LIN {X 0,Y 92.018,Z 344.154,A -85,B 0,C 180,E1 -28315.718,E2 -28315.718} C_VEL
LIN {X 0,Y 86.368,Z 354.698,A -85,B 0,C 180,E1 -28320.776,E2 -28320.776} C_VEL
LIN {X 0,Y 80.821,Z 363.839,A -85,B 0,C 180,E1 -28326.964,E2 -28326.964} C_VEL
LIN {X 0,Y 76.179,Z 371.216,A -85,B 0,C 180,E1 -28333.933,E2 -28333.933} C_VEL
LIN {X 0,Y 72.82,Z 377.117,A -85,B 0,C 180,E1 -28341.676,E2 -28341.676} C_VEL
LIN {X 0,Y 70.618,Z 381.782,A -85,B 0,C 180,E1 -28350,E2 -28350} C_VEL
LIN {X 0,Y 70.293,Z 382.581,A -85,B 0,C 180,E1 -28351.768,E2 -28351.768} C_VEL
LIN {X 0,Y 68.904,Z 384.476,A -85,B 0,C 180,E1 -28356.25,E2 -28356.25} C_VEL
LIN {X 0,Y 65.683,Z 386.983,A -85,B 0,C 180,E1 -28363.945,E2 -28363.945} C_VEL
LIN {X 0,Y 63.762,Z 388.494,A -85,B 0,C 180,E1 -28370.668,E2 -28370.668} C_VEL
LIN {X 0,Y 63.611,Z 389.367,A -85,B 0,C 180,E1 -28375.957,E2 -28375.957} C_VEL
LIN {X 0,Y 63.921,Z 389.596,A -85,B 0,C 180,E1 -28377.701,E2 -28377.701} C_VEL
LIN {X 0,Y 67.759,Z 390.402,A -85,B 0,C 180,E1 -28388.485,E2 -28388.485} C_VEL
LIN {X 0,Y 73.771,Z 389.834,A -85,B 0,C 180,E1 -28398.183,E2 -28398.183} C_VEL
LIN {X 0,Y 78.574,Z 388.718,A -85,B 0,C 180,E1 -28403.608,E2 -28403.608} C_VEL
LIN {X 0,Y 83.148,Z 387.318,A -85,B 0,C 180,E1 -28407.695,E2 -28407.695} C_VEL
LIN {X 0,Y 90.439,Z 384.448,A -85,B 0,C 180,E1 -28412.842,E2 -28412.842} C_VEL
LIN {X 0,Y 98.878,Z 380.236,A -85,B 0,C 180,E1 -28417.515,E2 -28417.515} C_VEL
LIN {X 0,Y 107.812,Z 374.74,A -85,B 0,C 180,E1 -28421.393,E2 -28421.393} C_VEL
LIN {X 0,Y 108.744,Z 373.558,A -85,B 0,C 180,E1 -28423.099,E2 -28423.099} C_VEL
LIN {X 0,Y 109.834,Z 371.724,A -85,B 0,C 180,E1 -28426.233,E2 -28426.233} C_VEL
LIN {X 0,Y 110.579,Z 370.301,A -85,B 0,C 180,E1 -28429.013,E2 -28429.013} C_VEL
LIN {X 0,Y 111.224,Z 368.711,A -85,B 0,C 180,E1 -28432.744,E2 -28432.744} C_VEL
LIN {X 0,Y 111.839,Z 367.436,A -85,B 0,C 180,E1 -28436.401,E2 -28436.401} C_VEL
LIN {X 0,Y 112.278,Z 366.529,A -85,B 0,C 180,E1 -28440.004,E2 -28440.004} C_VEL
LIN {X 0,Y 112.294,Z 366.253,A -85,B 0,C 180,E1 -28443.593,E2 -28443.593} C_VEL
LIN {X 0,Y 111.927,Z 366.629,A -85,B 0,C 180,E1 -28447.219,E2 -28447.219} C_VEL
LIN {X 0,Y 111.564,Z 367.372,A -85,B 0,C 180,E1 -28450.898,E2 -28450.898} C_VEL
LIN {X 0,Y 111.237,Z 368.424,A -85,B 0,C 180,E1 -28454.643,E2 -28454.643} C_VEL
LIN {X 0,Y 110.286,Z 370.941,A -85,B 0,C 180,E1 -28460.522,E2 -28460.522} C_VEL
LIN {X 0,Y 108.905,Z 373.784,A -85,B 0,C 180,E1 -28465.386,E2 -28465.386} C_VEL
LIN {X 0,Y 107.482,Z 376.257,A -85,B 0,C 180,E1 -28469.068,E2 -28469.068} C_VEL
LIN {X 0,Y 106.076,Z 377.68,A -85,B 0,C 180,E1 -28470.539,E2 -28470.539} C_VEL
LIN {X 0,Y 100.57,Z 381.248,A -85,B 0,C 180,E1 -28473.012,E2 -28473.012} C_VEL
LIN {X 0,Y 92.528,Z 385.67,A -85,B 0,C 180,E1 -28477.107,E2 -28477.107} C_VEL
LIN {X 0,Y 85.091,Z 389.05,A -85,B 0,C 180,E1 -28481.984,E2 -28481.984} C_VEL
LIN {X 0,Y 76.184,Z 392.05,A -85,B 0,C 180,E1 -28489.78,E2 -28489.78} C_VEL
LIN {X 0,Y 69.088,Z 393.493,A -85,B 0,C 180,E1 -28499.429,E2 -28499.429} C_VEL
LIN {X 0,Y 64.576,Z 393.358,A -85,B 0,C 180,E1 -28510.944,E2 -28510.944} C_VEL
LIN {X 0,Y 62.726,Z 391.712,A -85,B 0,C 180,E1 -28523.567,E2 -28523.567} C_VEL
LIN {X 0,Y 62.679,Z 390.242,A -85,B 0,C 180,E1 -28530,E2 -28530} C_VEL
LIN {X 0,Y 62.887,Z 387.196,A -85,B 0,C 180,E1 -28539.65,E2 -28539.65} C_VEL
LIN {X 0,Y 64.422,Z 383.057,A -85,B 0,C 180,E1 -28549.104,E2 -28549.104} C_VEL
LIN {X 0,Y 68.042,Z 376.693,A -85,B 0,C 180,E1 -28559.381,E2 -28559.381} C_VEL
LIN {X 0,Y 72.677,Z 369.751,A -85,B 0,C 180,E1 -28567.184,E2 -28567.184} C_VEL
LIN {X 0,Y 77.715,Z 361.895,A -85,B 0,C 180,E1 -28573.522,E2 -28573.522} C_VEL
LIN {X 0,Y 81.578,Z 355.857,A -85,B 0,C 180,E1 -28577.077,E2 -28577.077} C_VEL
LIN {X 0,Y 85.122,Z 346.402,A -85,B 0,C 180,E1 -28582.623,E2 -28582.623} C_VEL
LIN {X 0,Y 87.485,Z 337.692,A -85,B 0,C 180,E1 -28587.157,E2 -28587.157} C_VEL
LIN {X 0,Y 87.648,Z 335.398,A -85,B 0,C 180,E1 -28588.581,E2 -28588.581} C_VEL
LIN {X 0,Y 87.041,Z 330.108,A -85,B 0,C 180,E1 -28592.643,E2 -28592.643} C_VEL
LIN {X 0,Y 86.061,Z 326.798,A -85,B 0,C 180,E1 -28595.895,E2 -28595.895} C_VEL
LIN {X 0,Y 85.319,Z 324.626,A -85,B 0,C 180,E1 -28598.237,E2 -28598.237} C_VEL
LIN {X 0,Y 83.779,Z 321.175,A -85,B 0,C 180,E1 -28602.92,E2 -28602.92} C_VEL
LIN {X 0,Y 81.877,Z 316.988,A -85,B 0,C 180,E1 -28610.109,E2 -28610.109} C_VEL
LIN {X 0,Y 80.619,Z 314.216,A -85,B 0,C 180,E1 -28617.496,E2 -28617.496} C_VEL
LIN {X 0,Y 80.581,Z 313.017,A -85,B 0,C 180,E1 -28619.994,E2 -28619.994} C_VEL
LIN {X 0,Y 80.065,Z 312.777,A -85,B 0,C 180,E1 -28626.992,E2 -28626.992} C_VEL
LIN {X 0,Y 80.116,Z 312.914,A -85,B 0,C 180,E1 -28630.098,E2 -28630.098} C_VEL
LIN {X 0,Y 80.243,Z 314.44,A -85,B 0,C 180,E1 -28635.55,E2 -28635.55} C_VEL
LIN {X 0,Y 81.919,Z 317.887,A -85,B 0,C 180,E1 -28645.395,E2 -28645.395} C_VEL
LIN {X 0,Y 83.202,Z 320.714,A -85,B 0,C 180,E1 -28650.445,E2 -28650.445} C_VEL
LIN {X 0,Y 85.06,Z 325.54,A -85,B 0,C 180,E1 -28656.884,E2 -28656.884} C_VEL
LIN {X 0,Y 86.237,Z 328.978,A -85,B 0,C 180,E1 -28660.682,E2 -28660.682} C_VEL
LIN {X 0,Y 87.697,Z 334.701,A -85,B 0,C 180,E1 -28666.15,E2 -28666.15} C_VEL
LIN {X 0,Y 88.081,Z 336.72,A -85,B 0,C 180,E1 -28667.886,E2 -28667.886} C_VEL
LIN {X 0,Y 87.681,Z 340.216,A -85,B 0,C 180,E1 -28670.117,E2 -28670.117} C_VEL
LIN {X 0,Y 86.704,Z 344.364,A -85,B 0,C 180,E1 -28672.561,E2 -28672.561} C_VEL
LIN {X 0,Y 81.324,Z 353.994,A -85,B 0,C 180,E1 -28677.308,E2 -28677.308} C_VEL
LIN {X 0,Y 76.185,Z 361.944,A -85,B 0,C 180,E1 -28682.533,E2 -28682.533} C_VEL
LIN {X 0,Y 70.878,Z 369.719,A -85,B 0,C 180,E1 -28689.694,E2 -28689.694} C_VEL
LIN {X 0,Y 66.874,Z 375.937,A -85,B 0,C 180,E1 -28697.867,E2 -28697.867} C_VEL
LIN {X 0,Y 64.091,Z 380.892,A -85,B 0,C 180,E1 -28706.857,E2 -28706.857} C_VEL
LIN {X 0,Y 62.438,Z 384.742,A -85,B 0,C 180,E1 -28716.462,E2 -28716.462} C_VEL
LIN {X 0,Y 62.098,Z 386.739,A -85,B 0,C 180,E1 -28723.082,E2 -28723.082} C_VEL
LIN {X 0,Y 62.492,Z 388.303,A -85,B 0,C 180,E1 -28729.717,E2 -28729.717} C_VEL
LIN {X 0,Y 63.921,Z 389.596,A -85,B 0,C 180,E1 -28737.701,E2 -28737.701} C_VEL
LIN {X 0,Y 64.741,Z 390.181,A -85,B 0,C 180,E1 -28742.889,E2 -28742.889} C_VEL
LIN {X 0,Y 65.462,Z 390.63,A -85,B 0,C 180,E1 -28751.598,E2 -28751.598} C_VEL
LIN {X 0,Y 66.926,Z 390.437,A -85,B 0,C 180,E1 -28758.374,E2 -28758.374} C_VEL
LIN {X 0,Y 69.282,Z 389.92,A -85,B 0,C 180,E1 -28762.928,E2 -28762.928} C_VEL
LIN {X 0,Y 70.378,Z 389.67,A -85,B 0,C 180,E1 -28764.26,E2 -28764.26} C_VEL
LIN {X 0,Y 74.417,Z 388.783,A -85,B 0,C 180,E1 -28768.205,E2 -28768.205} C_VEL
LIN {X 0,Y 84.112,Z 385.635,A -85,B 0,C 180,E1 -28775.312,E2 -28775.312} C_VEL
LIN {X 0,Y 93.339,Z 381.565,A -85,B 0,C 180,E1 -28780.248,E2 -28780.248} C_VEL
LIN {X 0,Y 102.448,Z 376.503,A -85,B 0,C 180,E1 -28784.079,E2 -28784.079} C_VEL
LIN {X 0,Y 103.419,Z 375.35,A -85,B 0,C 180,E1 -28786.245,E2 -28786.245} C_VEL
LIN {X 0,Y 104.064,Z 374.379,A -85,B 0,C 180,E1 -28788.316,E2 -28788.316} C_VEL
LIN {X 0,Y 105.039,Z 372.811,A -85,B 0,C 180,E1 -28792.315,E2 -28792.315} C_VEL
LIN {X 0,Y 105.802,Z 371.552,A -85,B 0,C 180,E1 -28796.196,E2 -28796.196} C_VEL
LIN {X 0,Y 106.434,Z 370.677,A -85,B 0,C 180,E1 -28800.005,E2 -28800.005} C_VEL
LIN {X 0,Y 106.488,Z 370.442,A -85,B 0,C 180,E1 -28803.789,E2 -28803.789} C_VEL
LIN {X 0,Y 106.069,Z 370.864,A -85,B 0,C 180,E1 -28807.62,E2 -28807.62} C_VEL
LIN {X 0,Y 105.594,Z 371.64,A -85,B 0,C 180,E1 -28811.522,E2 -28811.522} C_VEL
LIN {X 0,Y 105.046,Z 372.775,A -85,B 0,C 180,E1 -28815.527,E2 -28815.527} C_VEL
LIN {X 0,Y 104.295,Z 374.396,A -85,B 0,C 180,E1 -28819.695,E2 -28819.695} C_VEL
LIN {X 0,Y 102.829,Z 376.705,A -85,B 0,C 180,E1 -28824.215,E2 -28824.215} C_VEL
LIN {X 0,Y 101.948,Z 377.966,A -85,B 0,C 180,E1 -28826.342,E2 -28826.342} C_VEL
LIN {X 0,Y 99.787,Z 379.719,A -85,B 0,C 180,E1 -28828.315,E2 -28828.315} C_VEL
LIN {X 0,Y 91.18,Z 384.423,A -85,B 0,C 180,E1 -28832.023,E2 -28832.023} C_VEL
LIN {X 0,Y 84.735,Z 387.375,A -85,B 0,C 180,E1 -28835.499,E2 -28835.499} C_VEL
LIN {X 0,Y 75.513,Z 390.701,A -85,B 0,C 180,E1 -28841.881,E2 -28841.881} C_VEL
LIN {X 0,Y 66.722,Z 392.85,A -85,B 0,C 180,E1 -28850.804,E2 -28850.804} C_VEL
LIN {X 0,Y 63.056,Z 393.309,A -85,B 0,C 180,E1 -28856.133,E2 -28856.133} C_VEL
LIN {X 0,Y 57.893,Z 393.106,A -85,B 0,C 180,E1 -28868.643,E2 -28868.643} C_VEL
LIN {X 0,Y 56.396,Z 392.443,A -85,B 0,C 180,E1 -28875.568,E2 -28875.568} C_VEL
LIN {X 0,Y 55.663,Z 391.363,A -85,B 0,C 180,E1 -28882.747,E2 -28882.747} C_VEL
LIN {X 0,Y 55.589,Z 389.853,A -85,B 0,C 180,E1 -28890,E2 -28890} C_VEL
LIN {X 0,Y 55.885,Z 386.73,A -85,B 0,C 180,E1 -28900.873,E2 -28900.873} C_VEL
LIN {X 0,Y 57.705,Z 382.508,A -85,B 0,C 180,E1 -28911.43,E2 -28911.43} C_VEL
LIN {X 0,Y 61.928,Z 376.062,A -85,B 0,C 180,E1 -28922.619,E2 -28922.619} C_VEL
LIN {X 0,Y 67.111,Z 369.001,A -85,B 0,C 180,E1 -28930.882,E2 -28930.882} C_VEL
LIN {X 0,Y 72.955,Z 360.676,A -85,B 0,C 180,E1 -28937.589,E2 -28937.589} C_VEL
LIN {X 0,Y 75.706,Z 356.698,A -85,B 0,C 180,E1 -28939.983,E2 -28939.983} C_VEL
LIN {X 0,Y 79.215,Z 348.739,A -85,B 0,C 180,E1 -28945.013,E2 -28945.013} C_VEL
LIN {X 0,Y 82.21,Z 339.886,A -85,B 0,C 180,E1 -28950.006,E2 -28950.006} C_VEL
LIN {X 0,Y 82.184,Z 335.431,A -85,B 0,C 180,E1 -28953.632,E2 -28953.632} C_VEL
LIN {X 0,Y 81.547,Z 331.959,A -85,B 0,C 180,E1 -28957.175,E2 -28957.175} C_VEL
LIN {X 0,Y 80.973,Z 329.88,A -85,B 0,C 180,E1 -28959.679,E2 -28959.679} C_VEL
LIN {X 0,Y 79.736,Z 326.561,A -85,B 0,C 180,E1 -28964.661,E2 -28964.661} C_VEL
LIN {X 0,Y 78.714,Z 323.787,A -85,B 0,C 180,E1 -28969.707,E2 -28969.707} C_VEL
LIN {X 0,Y 77.638,Z 319.844,A -85,B 0,C 180,E1 -28979.994,E2 -28979.994} C_VEL
LIN {X 0,Y 77.36,Z 319.227,A -85,B 0,C 180,E1 -28985.206,E2 -28985.206} C_VEL
LIN {X 0,Y 77.248,Z 319.631,A -85,B 0,C 180,E1 -28990.477,E2 -28990.477} C_VEL
LIN {X 0,Y 78.273,Z 323.727,A -85,B 0,C 180,E1 -29003.824,E2 -29003.824} C_VEL
LIN {X 0,Y 79.211,Z 326.244,A -85,B 0,C 180,E1 -29008.91,E2 -29008.91} C_VEL
LIN {X 0,Y 80.712,Z 331.117,A -85,B 0,C 180,E1 -29016.07,E2 -29016.07} C_VEL
LIN {X 0,Y 81.599,Z 334.606,A -85,B 0,C 180,E1 -29020.226,E2 -29020.226} C_VEL
LIN {X 0,Y 82.422,Z 339.119,A -85,B 0,C 180,E1 -29024.919,E2 -29024.919} C_VEL
LIN {X 0,Y 82.541,Z 340.301,A -85,B 0,C 180,E1 -29026.043,E2 -29026.043} C_VEL
LIN {X 0,Y 81.813,Z 343.621,A -85,B 0,C 180,E1 -29028.261,E2 -29028.261} C_VEL
LIN {X 0,Y 81.23,Z 345.605,A -85,B 0,C 180,E1 -29029.542,E2 -29029.542} C_VEL
LIN {X 0,Y 75.424,Z 355.068,A -85,B 0,C 180,E1 -29034.383,E2 -29034.383} C_VEL
LIN {X 0,Y 68.937,Z 364.216,A -85,B 0,C 180,E1 -29041.037,E2 -29041.037} C_VEL
LIN {X 0,Y 63.399,Z 371.597,A -85,B 0,C 180,E1 -29048.883,E2 -29048.883} C_VEL
LIN {X 0,Y 59.904,Z 376.587,A -85,B 0,C 180,E1 -29056.429,E2 -29056.429} C_VEL
LIN {X 0,Y 56.932,Z 381.448,A -85,B 0,C 180,E1 -29066.461,E2 -29066.461} C_VEL
LIN {X 0,Y 55.244,Z 385.213,A -85,B 0,C 180,E1 -29077.308,E2 -29077.308} C_VEL
LIN {X 0,Y 55.029,Z 387.169,A -85,B 0,C 180,E1 -29084.798,E2 -29084.798} C_VEL
LIN {X 0,Y 55.663,Z 388.654,A -85,B 0,C 180,E1 -29092.257,E2 -29092.257} C_VEL
LIN {X 0,Y 57.536,Z 389.922,A -85,B 0,C 180,E1 -29101.252,E2 -29101.252} C_VEL
LIN {X 0,Y 62.136,Z 390.62,A -85,B 0,C 180,E1 -29112.736,E2 -29112.736} C_VEL
LIN {X 0,Y 68.298,Z 390.08,A -85,B 0,C 180,E1 -29121.882,E2 -29121.882} C_VEL
LIN {X 0,Y 70.378,Z 389.67,A -85,B 0,C 180,E1 -29124.26,E2 -29124.26} C_VEL
LIN {X 0,Y 73.522,Z 388.919,A -85,B 0,C 180,E1 -29128.189,E2 -29128.189} C_VEL
LIN {X 0,Y 77.999,Z 387.228,A -85,B 0,C 180,E1 -29134.767,E2 -29134.767} C_VEL
LIN {X 0,Y 82.072,Z 385.454,A -85,B 0,C 180,E1 -29139.487,E2 -29139.487} C_VEL
LIN {X 0,Y 85.943,Z 383.765,A -85,B 0,C 180,E1 -29142.315,E2 -29142.315} C_VEL
LIN {X 0,Y 87.431,Z 383.121,A -85,B 0,C 180,E1 -29143.063,E2 -29143.063} C_VEL
LIN {X 0,Y 94.223,Z 379.862,A -85,B 0,C 180,E1 -29145.843,E2 -29145.843} C_VEL
LIN {X 0,Y 97.267,Z 378.117,A -85,B 0,C 180,E1 -29147.486,E2 -29147.486} C_VEL
LIN {X 0,Y 99.009,Z 376.01,A -85,B 0,C 180,E1 -29153.588,E2 -29153.588} C_VEL
LIN {X 0,Y 99.528,Z 375.344,A -85,B 0,C 180,E1 -29155.956,E2 -29155.956} C_VEL
LIN {X 0,Y 100.325,Z 374.473,A -85,B 0,C 180,E1 -29160.005,E2 -29160.005} C_VEL
LIN {X 0,Y 100.449,Z 374.273,A -85,B 0,C 180,E1 -29164.017,E2 -29164.017} C_VEL
LIN {X 0,Y 99.723,Z 374.978,A -85,B 0,C 180,E1 -29169.38,E2 -29169.38} C_VEL
LIN {X 0,Y 99.306,Z 375.582,A -85,B 0,C 180,E1 -29172.263,E2 -29172.263} C_VEL
LIN {X 0,Y 98.538,Z 376.825,A -85,B 0,C 180,E1 -29176.581,E2 -29176.581} C_VEL
LIN {X 0,Y 97.285,Z 378.592,A -85,B 0,C 180,E1 -29181.179,E2 -29181.179} C_VEL
LIN {X 0,Y 96.033,Z 380.11,A -85,B 0,C 180,E1 -29184.302,E2 -29184.302} C_VEL
LIN {X 0,Y 93.588,Z 381.569,A -85,B 0,C 180,E1 -29185.694,E2 -29185.694} C_VEL
LIN {X 0,Y 84.714,Z 385.821,A -85,B 0,C 180,E1 -29189.416,E2 -29189.416} C_VEL
LIN {X 0,Y 76.289,Z 389.043,A -85,B 0,C 180,E1 -29193.995,E2 -29193.995} C_VEL
LIN {X 0,Y 65.944,Z 391.894,A -85,B 0,C 180,E1 -29201.754,E2 -29201.754} C_VEL
LIN {X 0,Y 57.281,Z 393.126,A -85,B 0,C 180,E1 -29212.161,E2 -29212.161} C_VEL
LIN {X 0,Y 51.336,Z 392.854,A -85,B 0,C 180,E1 -29225.752,E2 -29225.752} C_VEL
LIN {X 0,Y 49.534,Z 392.146,A -85,B 0,C 180,E1 -29233.516,E2 -29233.516} C_VEL
LIN {X 0,Y 48.619,Z 391.008,A -85,B 0,C 180,E1 -29241.689,E2 -29241.689} C_VEL
LIN {X 0,Y 48.489,Z 389.462,A -85,B 0,C 180,E1 -29250,E2 -29250} C_VEL
LIN {X 0,Y 48.927,Z 386.265,A -85,B 0,C 180,E1 -29262.443,E2 -29262.443} C_VEL
LIN {X 0,Y 51.116,Z 381.961,A -85,B 0,C 180,E1 -29274.36,E2 -29274.36} C_VEL
LIN {X 0,Y 55.191,Z 376.447,A -85,B 0,C 180,E1 -29284.961,E2 -29284.961} C_VEL
LIN {X 0,Y 60.814,Z 369.536,A -85,B 0,C 180,E1 -29293.898,E2 -29293.898} C_VEL
LIN {X 0,Y 66.953,Z 361.573,A -85,B 0,C 180,E1 -29300.871,E2 -29300.871} C_VEL
LIN {X 0,Y 70.059,Z 357.537,A -85,B 0,C 180,E1 -29303.371,E2 -29303.371} C_VEL
LIN {X 0,Y 74.082,Z 349.648,A -85,B 0,C 180,E1 -29308.627,E2 -29308.627} C_VEL
LIN {X 0,Y 76.858,Z 342.723,A -85,B 0,C 180,E1 -29312.786,E2 -29312.786} C_VEL
LIN {X 0,Y 77.104,Z 339.462,A -85,B 0,C 180,E1 -29315.71,E2 -29315.71} C_VEL
LIN {X 0,Y 76.867,Z 336.939,A -85,B 0,C 180,E1 -29318.541,E2 -29318.541} C_VEL
LIN {X 0,Y 76.464,Z 334.946,A -85,B 0,C 180,E1 -29321.228,E2 -29321.228} C_VEL
LIN {X 0,Y 75.32,Z 331.184,A -85,B 0,C 180,E1 -29327.784,E2 -29327.784} C_VEL
LIN {X 0,Y 74.795,Z 329.245,A -85,B 0,C 180,E1 -29331.891,E2 -29331.891} C_VEL
LIN {X 0,Y 74.311,Z 326.374,A -85,B 0,C 180,E1 -29339.994,E2 -29339.994} C_VEL
LIN {X 0,Y 74.178,Z 325.607,A -85,B 0,C 180,E1 -29345.43,E2 -29345.43} C_VEL
LIN {X 0,Y 73.94,Z 326.198,A -85,B 0,C 180,E1 -29350.952,E2 -29350.952} C_VEL
LIN {X 0,Y 74.412,Z 329.43,A -85,B 0,C 180,E1 -29362.189,E2 -29362.189} C_VEL
LIN {X 0,Y 75.132,Z 331.917,A -85,B 0,C 180,E1 -29367.878,E2 -29367.878} C_VEL
LIN {X 0,Y 76.154,Z 336.478,A -85,B 0,C 180,E1 -29375.217,E2 -29375.217} C_VEL
LIN {X 0,Y 76.884,Z 341.5,A -85,B 0,C 180,E1 -29381.499,E2 -29381.499} C_VEL
LIN {X 0,Y 77.025,Z 342.964,A -85,B 0,C 180,E1 -29383.12,E2 -29383.12} C_VEL
LIN {X 0,Y 76.69,Z 344.858,A -85,B 0,C 180,E1 -29384.748,E2 -29384.748} C_VEL
LIN {X 0,Y 75.995,Z 346.846,A -85,B 0,C 180,E1 -29386.086,E2 -29386.086} C_VEL
LIN {X 0,Y 69.755,Z 356.083,A -85,B 0,C 180,E1 -29390.973,E2 -29390.973} C_VEL
LIN {X 0,Y 62.809,Z 365.084,A -85,B 0,C 180,E1 -29397.893,E2 -29397.893} C_VEL
LIN {X 0,Y 56.826,Z 372.347,A -85,B 0,C 180,E1 -29406.301,E2 -29406.301} C_VEL
LIN {X 0,Y 52.968,Z 377.238,A -85,B 0,C 180,E1 -29414.611,E2 -29414.611} C_VEL
LIN {X 0,Y 49.856,Z 381.832,A -85,B 0,C 180,E1 -29425.472,E2 -29425.472} C_VEL
LIN {X 0,Y 48.038,Z 385.686,A -85,B 0,C 180,E1 -29438.412,E2 -29438.412} C_VEL
LIN {X 0,Y 48.007,Z 387.582,A -85,B 0,C 180,E1 -29447.024,E2 -29447.024} C_VEL
LIN {X 0,Y 48.978,Z 389,A -85,B 0,C 180,E1 -29455.497,E2 -29455.497} C_VEL
LIN {X 0,Y 50.96,Z 390.081,A -85,B 0,C 180,E1 -29464.177,E2 -29464.177} C_VEL
LIN {X 0,Y 53.496,Z 390.637,A -85,B 0,C 180,E1 -29471.06,E2 -29471.06} C_VEL
LIN {X 0,Y 56.919,Z 390.811,A -85,B 0,C 180,E1 -29477.801,E2 -29477.801} C_VEL
LIN {X 0,Y 64.901,Z 390.038,A -85,B 0,C 180,E1 -29488.071,E2 -29488.071} C_VEL
LIN {X 0,Y 70.798,Z 388.842,A -85,B 0,C 180,E1 -29493.302,E2 -29493.302} C_VEL
LIN {X 0,Y 80.315,Z 385.947,A -85,B 0,C 180,E1 -29499.518,E2 -29499.518} C_VEL
LIN {X 0,Y 87.431,Z 383.121,A -85,B 0,C 180,E1 -29503.063,E2 -29503.063} C_VEL
LIN {X 0,Y 89.562,Z 382.105,A -85,B 0,C 180,E1 -29504.516,E2 -29504.516} C_VEL
LIN {X 0,Y 91.378,Z 380.923,A -85,B 0,C 180,E1 -29507.122,E2 -29507.122} C_VEL
LIN {X 0,Y 92.343,Z 379.9,A -85,B 0,C 180,E1 -29510.498,E2 -29510.498} C_VEL
LIN {X 0,Y 93.08,Z 378.754,A -85,B 0,C 180,E1 -29515.833,E2 -29515.833} C_VEL
LIN {X 0,Y 94.012,Z 377.933,A -85,B 0,C 180,E1 -29520.005,E2 -29520.005} C_VEL
LIN {X 0,Y 94.147,Z 377.776,A -85,B 0,C 180,E1 -29524.286,E2 -29524.286} C_VEL
LIN {X 0,Y 93.564,Z 378.28,A -85,B 0,C 180,E1 -29528.645,E2 -29528.645} C_VEL
LIN {X 0,Y 92.725,Z 379.216,A -85,B 0,C 180,E1 -29533.148,E2 -29533.148} C_VEL
LIN {X 0,Y 91.591,Z 380.548,A -85,B 0,C 180,E1 -29537.88,E2 -29537.88} C_VEL
LIN {X 0,Y 90.446,Z 381.749,A -85,B 0,C 180,E1 -29541.184,E2 -29541.184} C_VEL
LIN {X 0,Y 87.595,Z 383.238,A -85,B 0,C 180,E1 -29542.683,E2 -29542.683} C_VEL
LIN {X 0,Y 75.767,Z 388.019,A -85,B 0,C 180,E1 -29547.639,E2 -29547.639} C_VEL
LIN {X 0,Y 66.87,Z 390.626,A -85,B 0,C 180,E1 -29552.779,E2 -29552.779} C_VEL
LIN {X 0,Y 61.43,Z 391.803,A -85,B 0,C 180,E1 -29556.791,E2 -29556.791} C_VEL
LIN {X 0,Y 51.846,Z 392.943,A -85,B 0,C 180,E1 -29567.332,E2 -29567.332} C_VEL
LIN {X 0,Y 44.936,Z 392.599,A -85,B 0,C 180,E1 -29582.019,E2 -29582.019} C_VEL
LIN {X 0,Y 42.767,Z 391.824,A -85,B 0,C 180,E1 -29590.813,E2 -29590.813} C_VEL
LIN {X 0,Y 41.61,Z 390.648,A -85,B 0,C 180,E1 -29600.277,E2 -29600.277} C_VEL
LIN {X 0,Y 41.407,Z 389.068,A -85,B 0,C 180,E1 -29610,E2 -29610} C_VEL
LIN {X 0,Y 42.004,Z 385.793,A -85,B 0,C 180,E1 -29624.535,E2 -29624.535} C_VEL
LIN {X 0,Y 44.711,Z 381.406,A -85,B 0,C 180,E1 -29638.136,E2 -29638.136} C_VEL
LIN {X 0,Y 49.515,Z 375.802,A -85,B 0,C 180,E1 -29649.695,E2 -29649.695} C_VEL
LIN {X 0,Y 55.879,Z 368.781,A -85,B 0,C 180,E1 -29658.992,E2 -29658.992} C_VEL
LIN {X 0,Y 62.714,Z 360.654,A -85,B 0,C 180,E1 -29665.913,E2 -29665.913} C_VEL
LIN {X 0,Y 65.905,Z 356.508,A -85,B 0,C 180,E1 -29668.55,E2 -29668.55} C_VEL
LIN {X 0,Y 70.271,Z 348.361,A -85,B 0,C 180,E1 -29674.171,E2 -29674.171} C_VEL
LIN {X 0,Y 71.734,Z 345.243,A -85,B 0,C 180,E1 -29676.156,E2 -29676.156} C_VEL
LIN {X 0,Y 72.015,Z 341.752,A -85,B 0,C 180,E1 -29680.021,E2 -29680.021} C_VEL
LIN {X 0,Y 71.778,Z 339.866,A -85,B 0,C 180,E1 -29682.911,E2 -29682.911} C_VEL
LIN {X 0,Y 71.161,Z 336.849,A -85,B 0,C 180,E1 -29688.601,E2 -29688.601} C_VEL
LIN {X 0,Y 70.729,Z 334.539,A -85,B 0,C 180,E1 -29694.291,E2 -29694.291} C_VEL
LIN {X 0,Y 70.622,Z 332.684,A -85,B 0,C 180,E1 -29699.993,E2 -29699.993} C_VEL
LIN {X 0,Y 70.594,Z 331.831,A -85,B 0,C 180,E1 -29705.707,E2 -29705.707} C_VEL
LIN {X 0,Y 70.242,Z 332.615,A -85,B 0,C 180,E1 -29711.536,E2 -29711.536} C_VEL
LIN {X 0,Y 70.154,Z 334.157,A -85,B 0,C 180,E1 -29717.483,E2 -29717.483} C_VEL
LIN {X 0,Y 70.503,Z 336.067,A -85,B 0,C 180,E1 -29723.492,E2 -29723.492} C_VEL
LIN {X 0,Y 70.812,Z 337.375,A -85,B 0,C 180,E1 -29726.719,E2 -29726.719} C_VEL
LIN {X 0,Y 71.314,Z 341.288,A -85,B 0,C 180,E1 -29733.717,E2 -29733.717} C_VEL
LIN {X 0,Y 71.547,Z 345.862,A -85,B 0,C 180,E1 -29740.074,E2 -29740.074} C_VEL
LIN {X 0,Y 71.441,Z 347.015,A -85,B 0,C 180,E1 -29741.347,E2 -29741.347} C_VEL
LIN {X 0,Y 70.929,Z 348.192,A -85,B 0,C 180,E1 -29742.235,E2 -29742.235} C_VEL
LIN {X 0,Y 64.359,Z 357.055,A -85,B 0,C 180,E1 -29746.961,E2 -29746.961} C_VEL
LIN {X 0,Y 56.902,Z 365.925,A -85,B 0,C 180,E1 -29754.079,E2 -29754.079} C_VEL
LIN {X 0,Y 50.406,Z 373.046,A -85,B 0,C 180,E1 -29763.055,E2 -29763.055} C_VEL
LIN {X 0,Y 46.108,Z 377.869,A -85,B 0,C 180,E1 -29772.251,E2 -29772.251} C_VEL
LIN {X 0,Y 42.198,Z 383.18,A -85,B 0,C 180,E1 -29787.528,E2 -29787.528} C_VEL
LIN {X 0,Y 40.849,Z 386.148,A -85,B 0,C 180,E1 -29799.906,E2 -29799.906} C_VEL
LIN {X 0,Y 41.08,Z 387.964,A -85,B 0,C 180,E1 -29810.008,E2 -29810.008} C_VEL
LIN {X 0,Y 42.461,Z 389.344,A -85,B 0,C 180,E1 -29819.771,E2 -29819.771} C_VEL
LIN {X 0,Y 44.843,Z 390.323,A -85,B 0,C 180,E1 -29828.819,E2 -29828.819} C_VEL
LIN {X 0,Y 48.176,Z 390.886,A -85,B 0,C 180,E1 -29836.835,E2 -29836.835} C_VEL
LIN {X 0,Y 52.243,Z 390.999,A -85,B 0,C 180,E1 -29843.815,E2 -29843.815} C_VEL
LIN {X 0,Y 58.399,Z 390.576,A -85,B 0,C 180,E1 -29851.234,E2 -29851.234} C_VEL
LIN {X 0,Y 67.793,Z 388.874,A -85,B 0,C 180,E1 -29858.905,E2 -29858.905} C_VEL
LIN {X 0,Y 77.039,Z 386.243,A -85,B 0,C 180,E1 -29864.123,E2 -29864.123} C_VEL
LIN {X 0,Y 86.203,Z 382.734,A -85,B 0,C 180,E1 -29868.045,E2 -29868.045} C_VEL
LIN {X 0,Y 89.083,Z 381.438,A -85,B 0,C 180,E1 -29869.086,E2 -29869.086} C_VEL
LIN {X 0,Y 91.691,Z 379.981,A -85,B 0,C 180,E1 -29871.187,E2 -29871.187} C_VEL
LIN {X 0,Y 93.08,Z 378.754,A -85,B 0,C 180,E1 -29875.833,E2 -29875.833} C_VEL
LIN {X 0,Y 93.082,Z 378.529,A -85,B 0,C 180,E1 -29878.235,E2 -29878.235} C_VEL
LIN {X 0,Y 92.023,Z 378.891,A -85,B 0,C 180,E1 -29881.829,E2 -29881.829} C_VEL
LIN {X 0,Y 90.232,Z 379.768,A -85,B 0,C 180,E1 -29885.378,E2 -29885.378} C_VEL
LIN {X 0,Y 85.418,Z 382.839,A -85,B 0,C 180,E1 -29895.667,E2 -29895.667} C_VEL
LIN {X 0,Y 85.265,Z 383.002,A -85,B 0,C 180,E1 -29896.384,E2 -29896.384} C_VEL
LIN {X 0,Y 83.947,Z 383.871,A -85,B 0,C 180,E1 -29898.617,E2 -29898.617} C_VEL
LIN {X 0,Y 71.987,Z 388.27,A -85,B 0,C 180,E1 -29902.994,E2 -29902.994} C_VEL
LIN {X 0,Y 63.297,Z 390.586,A -85,B 0,C 180,E1 -29907.349,E2 -29907.349} C_VEL
LIN {X 0,Y 51.965,Z 392.415,A -85,B 0,C 180,E1 -29915.763,E2 -29915.763} C_VEL
LIN {X 0,Y 42.4,Z 392.737,A -85,B 0,C 180,E1 -29928.472,E2 -29928.472} C_VEL
LIN {X 0,Y 38.777,Z 392.323,A -85,B 0,C 180,E1 -29937.064,E2 -29937.064} C_VEL
LIN {X 0,Y 36.139,Z 391.498,A -85,B 0,C 180,E1 -29947.112,E2 -29947.112} C_VEL
LIN {X 0,Y 34.649,Z 390.286,A -85,B 0,C 180,E1 -29958.298,E2 -29958.298} C_VEL
LIN {X 0,Y 34.308,Z 388.668,A -85,B 0,C 180,E1 -29970.001,E2 -29970.001} C_VEL
LIN {X 0,Y 35.141,Z 385.312,A -85,B 0,C 180,E1 -29987.457,E2 -29987.457} C_VEL
LIN {X 0,Y 38.567,Z 380.842,A -85,B 0,C 180,E1 -30003.139,E2 -30003.139} C_VEL
LIN {X 0,Y 44.268,Z 375.148,A -85,B 0,C 180,E1 -30015.594,E2 -30015.594} C_VEL
LIN {X 0,Y 51.471,Z 367.975,A -85,B 0,C 180,E1 -30025.009,E2 -30025.009} C_VEL
LIN {X 0,Y 58.046,Z 360.8,A -85,B 0,C 180,E1 -30031.024,E2 -30031.024} C_VEL
LIN {X 0,Y 61.037,Z 357.315,A -85,B 0,C 180,E1 -30033.166,E2 -30033.166} C_VEL
LIN {X 0,Y 65.606,Z 349.908,A -85,B 0,C 180,E1 -30038.48,E2 -30038.48} C_VEL
LIN {X 0,Y 66.76,Z 347.724,A -85,B 0,C 180,E1 -30039.986,E2 -30039.986} C_VEL
LIN {X 0,Y 66.965,Z 346.437,A -85,B 0,C 180,E1 -30041.641,E2 -30041.641} C_VEL
LIN {X 0,Y 66.96,Z 344.575,A -85,B 0,C 180,E1 -30044.78,E2 -30044.78} C_VEL
LIN {X 0,Y 66.601,Z 340.58,A -85,B 0,C 180,E1 -30053.935,E2 -30053.935} C_VEL
LIN {X 0,Y 66.603,Z 338.76,A -85,B 0,C 180,E1 -30059.993,E2 -30059.993} C_VEL
LIN {X 0,Y 66.636,Z 337.903,A -85,B 0,C 180,E1 -30066.193,E2 -30066.193} C_VEL
LIN {X 0,Y 66.195,Z 338.825,A -85,B 0,C 180,E1 -30072.252,E2 -30072.252} C_VEL
LIN {X 0,Y 66.096,Z 341.349,A -85,B 0,C 180,E1 -30081.841,E2 -30081.841} C_VEL
LIN {X 0,Y 66.262,Z 342.484,A -85,B 0,C 180,E1 -30085.095,E2 -30085.095} C_VEL
LIN {X 0,Y 66.319,Z 345.932,A -85,B 0,C 180,E1 -30092.031,E2 -30092.031} C_VEL
LIN {X 0,Y 66.215,Z 348.55,A -85,B 0,C 180,E1 -30096.232,E2 -30096.232} C_VEL
LIN {X 0,Y 65.948,Z 349.904,A -85,B 0,C 180,E1 -30097.994,E2 -30097.994} C_VEL
LIN {X 0,Y 57.961,Z 359.643,A -85,B 0,C 180,E1 -30103.322,E2 -30103.322} C_VEL
LIN {X 0,Y 49.976,Z 368.005,A -85,B 0,C 180,E1 -30110.742,E2 -30110.742} C_VEL
LIN {X 0,Y 43.143,Z 374.734,A -85,B 0,C 180,E1 -30120.745,E2 -30120.745} C_VEL
LIN {X 0,Y 37.832,Z 380.118,A -85,B 0,C 180,E1 -30133.82,E2 -30133.82} C_VEL
LIN {X 0,Y 34.549,Z 384.342,A -85,B 0,C 180,E1 -30149.999,E2 -30149.999} C_VEL
LIN {X 0,Y 33.692,Z 386.591,A -85,B 0,C 180,E1 -30162.039,E2 -30162.039} C_VEL
LIN {X 0,Y 34.298,Z 388.345,A -85,B 0,C 180,E1 -30174.192,E2 -30174.192} C_VEL
LIN {X 0,Y 38.447,Z 390.4,A -85,B 0,C 180,E1 -30193.034,E2 -30193.034} C_VEL
LIN {X 0,Y 43.452,Z 391.114,A -85,B 0,C 180,E1 -30203.968,E2 -30203.968} C_VEL
LIN {X 0,Y 48.245,Z 391.187,A -85,B 0,C 180,E1 -30210.928,E2 -30210.928} C_VEL
LIN {X 0,Y 54.197,Z 390.812,A -85,B 0,C 180,E1 -30217.116,E2 -30217.116} C_VEL
LIN {X 0,Y 59.405,Z 390.115,A -85,B 0,C 180,E1 -30221.161,E2 -30221.161} C_VEL
LIN {X 0,Y 65.492,Z 388.904,A -85,B 0,C 180,E1 -30224.964,E2 -30224.964} C_VEL
LIN {X 0,Y 74.229,Z 386.563,A -85,B 0,C 180,E1 -30229.091,E2 -30229.091} C_VEL
LIN {X 0,Y 84.979,Z 382.593,A -85,B 0,C 180,E1 -30232.933,E2 -30232.933} C_VEL
LIN {X 0,Y 86.291,Z 381.847,A -85,B 0,C 180,E1 -30235.334,E2 -30235.334} C_VEL
LIN {X 0,Y 87.472,Z 381.069,A -85,B 0,C 180,E1 -30240.006,E2 -30240.006} C_VEL
LIN {X 0,Y 87.643,Z 380.943,A -85,B 0,C 180,E1 -30244.605,E2 -30244.605} C_VEL
LIN {X 0,Y 86.961,Z 381.49,A -85,B 0,C 180,E1 -30249.307,E2 -30249.307} C_VEL
LIN {X 0,Y 86.335,Z 382.062,A -85,B 0,C 180,E1 -30252.361,E2 -30252.361} C_VEL
LIN {X 0,Y 85.418,Z 382.839,A -85,B 0,C 180,E1 -30255.667,E2 -30255.667} C_VEL
LIN {X 0,Y 84.339,Z 383.46,A -85,B 0,C 180,E1 -30256.939,E2 -30256.939} C_VEL
LIN {X 0,Y 81.865,Z 384.547,A -85,B 0,C 180,E1 -30257.886,E2 -30257.886} C_VEL
LIN {X 0,Y 77.579,Z 386.061,A -85,B 0,C 180,E1 -30258.317,E2 -30258.317} C_VEL
LIN {X 0,Y 70,Z 388.233,A -85,B 0,C 180,E1 -30258.181,E2 -30258.181} C_VEL
LIN {X 0,Y 65.611,Z 389.301,A -85,B 0,C 180,E1 -30259.034,E2 -30259.034} C_VEL
LIN {X 0,Y 54.119,Z 391.583,A -85,B 0,C 180,E1 -30264.633,E2 -30264.633} C_VEL
LIN {X 0,Y 42.5,Z 392.579,A -85,B 0,C 180,E1 -30274.23,E2 -30274.23} C_VEL
LIN {X 0,Y 37.36,Z 392.512,A -85,B 0,C 180,E1 -30281.199,E2 -30281.199} C_VEL
LIN {X 0,Y 29.703,Z 391.171,A -85,B 0,C 180,E1 -30301.758,E2 -30301.758} C_VEL
LIN {X 0,Y 27.735,Z 389.923,A -85,B 0,C 180,E1 -30315.322,E2 -30315.322} C_VEL
LIN {X 0,Y 27.224,Z 388.267,A -85,B 0,C 180,E1 -30330.001,E2 -30330.001} C_VEL
LIN {X 0,Y 28.428,Z 384.832,A -85,B 0,C 180,E1 -30351.767,E2 -30351.767} C_VEL
LIN {X 0,Y 32.816,Z 380.275,A -85,B 0,C 180,E1 -30369.977,E2 -30369.977} C_VEL
LIN {X 0,Y 40.897,Z 373.341,A -85,B 0,C 180,E1 -30384.712,E2 -30384.712} C_VEL
LIN {X 0,Y 49.048,Z 365.883,A -85,B 0,C 180,E1 -30393.247,E2 -30393.247} C_VEL
LIN {X 0,Y 56.627,Z 358.06,A -85,B 0,C 180,E1 -30398.553,E2 -30398.553} C_VEL
LIN {X 0,Y 61.213,Z 351.579,A -85,B 0,C 180,E1 -30403.289,E2 -30403.289} C_VEL
LIN {X 0,Y 61.868,Z 350.323,A -85,B 0,C 180,E1 -30404.508,E2 -30404.508} C_VEL
LIN {X 0,Y 62.001,Z 349.104,A -85,B 0,C 180,E1 -30406.889,E2 -30406.889} C_VEL
LIN {X 0,Y 62.033,Z 346.468,A -85,B 0,C 180,E1 -30413.487,E2 -30413.487} C_VEL
LIN {X 0,Y 62.23,Z 344.6,A -85,B 0,C 180,E1 -30419.992,E2 -30419.992} C_VEL
LIN {X 0,Y 62.366,Z 343.742,A -85,B 0,C 180,E1 -30426.463,E2 -30426.463} C_VEL
LIN {X 0,Y 61.754,Z 344.8,A -85,B 0,C 180,E1 -30433.149,E2 -30433.149} C_VEL
LIN {X 0,Y 61.502,Z 346.449,A -85,B 0,C 180,E1 -30440.04,E2 -30440.04} C_VEL
LIN {X 0,Y 61.51,Z 347.666,A -85,B 0,C 180,E1 -30443.928,E2 -30443.928} C_VEL
LIN {X 0,Y 61.224,Z 350.131,A -85,B 0,C 180,E1 -30449.569,E2 -30449.569} C_VEL
LIN {X 0,Y 61.065,Z 351.385,A -85,B 0,C 180,E1 -30451.958,E2 -30451.958} C_VEL
LIN {X 0,Y 60.567,Z 352.58,A -85,B 0,C 180,E1 -30453.506,E2 -30453.506} C_VEL
LIN {X 0,Y 51.876,Z 362.035,A -85,B 0,C 180,E1 -30458.833,E2 -30458.833} C_VEL
LIN {X 0,Y 43.33,Z 370.023,A -85,B 0,C 180,E1 -30466.422,E2 -30466.422} C_VEL
LIN {X 0,Y 37.086,Z 375.411,A -85,B 0,C 180,E1 -30475.353,E2 -30475.353} C_VEL
LIN {X 0,Y 31.031,Z 380.701,A -85,B 0,C 180,E1 -30490.14,E2 -30490.14} C_VEL
LIN {X 0,Y 27.282,Z 384.846,A -85,B 0,C 180,E1 -30509.999,E2 -30509.999} C_VEL
LIN {X 0,Y 26.626,Z 387.011,A -85,B 0,C 180,E1 -30525.303,E2 -30525.303} C_VEL
LIN {X 0,Y 27.79,Z 388.726,A -85,B 0,C 180,E1 -30540.382,E2 -30540.382} C_VEL
LIN {X 0,Y 32.739,Z 390.56,A -85,B 0,C 180,E1 -30559.928,E2 -30559.928} C_VEL
LIN {X 0,Y 39.557,Z 391.341,A -85,B 0,C 180,E1 -30572.661,E2 -30572.661} C_VEL
LIN {X 0,Y 50.715,Z 391.04,A -85,B 0,C 180,E1 -30583.92,E2 -30583.92} C_VEL
LIN {X 0,Y 57.445,Z 390.187,A -85,B 0,C 180,E1 -30588.16,E2 -30588.16} C_VEL
LIN {X 0,Y 63.974,Z 388.934,A -85,B 0,C 180,E1 -30591.373,E2 -30591.373} C_VEL
LIN {X 0,Y 71.992,Z 386.89,A -85,B 0,C 180,E1 -30594.405,E2 -30594.405} C_VEL
LIN {X 0,Y 77.485,Z 385.114,A -85,B 0,C 180,E1 -30596.101,E2 -30596.101} C_VEL
LIN {X 0,Y 80.194,Z 384.07,A -85,B 0,C 180,E1 -30598.121,E2 -30598.121} C_VEL
LIN {X 0,Y 80.748,Z 383.824,A -85,B 0,C 180,E1 -30600.006,E2 -30600.006} C_VEL
LIN {X 0,Y 80.948,Z 383.758,A -85,B 0,C 180,E1 -30604.987,E2 -30604.987} C_VEL
LIN {X 0,Y 80.091,Z 384.33,A -85,B 0,C 180,E1 -30610.114,E2 -30610.114} C_VEL
LIN {X 0,Y 79.001,Z 384.997,A -85,B 0,C 180,E1 -30613.454,E2 -30613.454} C_VEL
LIN {X 0,Y 78.168,Z 385.434,A -85,B 0,C 180,E1 -30614.874,E2 -30614.874} C_VEL
LIN {X 0,Y 65.611,Z 389.301,A -85,B 0,C 180,E1 -30619.034,E2 -30619.034} C_VEL
LIN {X 0,Y 60.112,Z 390.517,A -85,B 0,C 180,E1 -30620.738,E2 -30620.738} C_VEL
LIN {X 0,Y 50.422,Z 391.838,A -85,B 0,C 180,E1 -30622.502,E2 -30622.502} C_VEL
LIN {X 0,Y 42.635,Z 392.321,A -85,B 0,C 180,E1 -30624.362,E2 -30624.362} C_VEL
LIN {X 0,Y 37.118,Z 392.383,A -85,B 0,C 180,E1 -30627.43,E2 -30627.43} C_VEL
LIN {X 0,Y 35.434,Z 392.318,A -85,B 0,C 180,E1 -30629.047,E2 -30629.047} C_VEL
LIN {X 0,Y 27.908,Z 391.742,A -85,B 0,C 180,E1 -30640.936,E2 -30640.936} C_VEL
LIN {X 0,Y 20.934,Z 389.561,A -85,B 0,C 180,E1 -30670.385,E2 -30670.385} C_VEL
LIN {X 0,Y 20.117,Z 387.842,A -85,B 0,C 180,E1 -30690.001,E2 -30690.001} C_VEL
LIN {X 0,Y 21.983,Z 384.335,A -85,B 0,C 180,E1 -30718.657,E2 -30718.657} C_VEL
LIN {X 0,Y 27.713,Z 379.68,A -85,B 0,C 180,E1 -30739.535,E2 -30739.535} C_VEL
LIN {X 0,Y 37.229,Z 372.637,A -85,B 0,C 180,E1 -30753.725,E2 -30753.725} C_VEL
LIN {X 0,Y 46.061,Z 365.231,A -85,B 0,C 180,E1 -30761.127,E2 -30761.127} C_VEL
LIN {X 0,Y 52.789,Z 358.768,A -85,B 0,C 180,E1 -30764.839,E2 -30764.839} C_VEL
LIN {X 0,Y 56.187,Z 354.669,A -85,B 0,C 180,E1 -30767.757,E2 -30767.757} C_VEL
LIN {X 0,Y 56.918,Z 353.448,A -85,B 0,C 180,E1 -30769.321,E2 -30769.321} C_VEL
LIN {X 0,Y 57.254,Z 351.082,A -85,B 0,C 180,E1 -30776.473,E2 -30776.473} C_VEL
LIN {X 0,Y 57.481,Z 350.181,A -85,B 0,C 180,E1 -30779.992,E2 -30779.992} C_VEL
LIN {X 0,Y 57.671,Z 349.38,A -85,B 0,C 180,E1 -30786.991,E2 -30786.991} C_VEL
LIN {X 0,Y 56.923,Z 350.571,A -85,B 0,C 180,E1 -30794.287,E2 -30794.287} C_VEL
LIN {X 0,Y 56.585,Z 352.362,A -85,B 0,C 180,E1 -30801.867,E2 -30801.867} C_VEL
LIN {X 0,Y 55.742,Z 354.95,A -85,B 0,C 180,E1 -30808.048,E2 -30808.048} C_VEL
LIN {X 0,Y 47.738,Z 362.935,A -85,B 0,C 180,E1 -30812.167,E2 -30812.167} C_VEL
LIN {X 0,Y 38.487,Z 370.764,A -85,B 0,C 180,E1 -30819.097,E2 -30819.097} C_VEL
LIN {X 0,Y 31.484,Z 376.085,A -85,B 0,C 180,E1 -30827.958,E2 -30827.958} C_VEL
LIN {X 0,Y 24.421,Z 381.271,A -85,B 0,C 180,E1 -30844.425,E2 -30844.425} C_VEL
LIN {X 0,Y 20.016,Z 385.331,A -85,B 0,C 180,E1 -30869.999,E2 -30869.999} C_VEL
LIN {X 0,Y 19.679,Z 387.433,A -85,B 0,C 180,E1 -30890.922,E2 -30890.922} C_VEL
LIN {X 0,Y 21.806,Z 389.108,A -85,B 0,C 180,E1 -30910.133,E2 -30910.133} C_VEL
LIN {X 0,Y 27.653,Z 390.716,A -85,B 0,C 180,E1 -30929.47,E2 -30929.47} C_VEL
LIN {X 0,Y 36.748,Z 391.569,A -85,B 0,C 180,E1 -30942.98,E2 -30942.98} C_VEL
LIN {X 0,Y 47.997,Z 391.271,A -85,B 0,C 180,E1 -30951.59,E2 -30951.59} C_VEL
LIN {X 0,Y 56.392,Z 390.257,A -85,B 0,C 180,E1 -30955.549,E2 -30955.549} C_VEL
LIN {X 0,Y 63.289,Z 388.965,A -85,B 0,C 180,E1 -30958,E2 -30958} C_VEL
LIN {X 0,Y 72.033,Z 386.72,A -85,B 0,C 180,E1 -30960.384,E2 -30960.384} C_VEL
LIN {X 0,Y 74.029,Z 386.109,A -85,B 0,C 180,E1 -30961.55,E2 -30961.55} C_VEL
LIN {X 0,Y 74.036,Z 386.166,A -85,B 0,C 180,E1 -30965.454,E2 -30965.454} C_VEL
LIN {X 0,Y 73.606,Z 386.396,A -85,B 0,C 180,E1 -30968.012,E2 -30968.012} C_VEL
LIN {X 0,Y 71.56,Z 387.174,A -85,B 0,C 180,E1 -30970.86,E2 -30970.86} C_VEL
LIN {X 0,Y 63.009,Z 389.417,A -85,B 0,C 180,E1 -30973.154,E2 -30973.154} C_VEL
LIN {X 0,Y 51.562,Z 391.473,A -85,B 0,C 180,E1 -30977.43,E2 -30977.43} C_VEL
LIN {X 0,Y 38.951,Z 392.397,A -85,B 0,C 180,E1 -30985.56,E2 -30985.56} C_VEL
LIN {X 0,Y 35.434,Z 392.318,A -85,B 0,C 180,E1 -30989.047,E2 -30989.047} C_VEL
LIN {X 0,Y 30.373,Z 392.066,A -85,B 0,C 180,E1 -30994.336,E2 -30994.336} C_VEL
LIN {X 0,Y 21.705,Z 390.885,A -85,B 0,C 180,E1 -31004.707,E2 -31004.707} C_VEL
LIN {X 0,Y 15.641,Z 389.398,A -85,B 0,C 180,E1 -31020.184,E2 -31020.184} C_VEL
LIN {X 0,Y 13.128,Z 387.971,A -85,B 0,C 180,E1 -31041.152,E2 -31041.152} C_VEL
LIN {X 0,Y 13.007,Z 387.427,A -85,B 0,C 180,E1 -31049.59,E2 -31049.59} C_VEL
LIN {X 0,Y 16.088,Z 383.814,A -85,B 0,C 180,E1 -31090.94,E2 -31090.94} C_VEL
LIN {X 0,Y 23.702,Z 379.07,A -85,B 0,C 180,E1 -31112.817,E2 -31112.817} C_VEL
LIN {X 0,Y 34.665,Z 371.933,A -85,B 0,C 180,E1 -31124.368,E2 -31124.368} C_VEL
LIN {X 0,Y 44.646,Z 364.037,A -85,B 0,C 180,E1 -31130.236,E2 -31130.236} C_VEL
LIN {X 0,Y 49.675,Z 359.476,A -85,B 0,C 180,E1 -31132.028,E2 -31132.028} C_VEL
LIN {X 0,Y 50.843,Z 358.277,A -85,B 0,C 180,E1 -31132.738,E2 -31132.738} C_VEL
LIN {X 0,Y 51.932,Z 356.965,A -85,B 0,C 180,E1 -31134.288,E2 -31134.288} C_VEL
LIN {X 0,Y 52.438,Z 355.48,A -85,B 0,C 180,E1 -31139.991,E2 -31139.991} C_VEL
LIN {X 0,Y 52.644,Z 354.758,A -85,B 0,C 180,E1 -31147.663,E2 -31147.663} C_VEL
LIN {X 0,Y 51.578,Z 356.501,A -85,B 0,C 180,E1 -31157.483,E2 -31157.483} C_VEL
LIN {X 0,Y 50.969,Z 357.75,A -85,B 0,C 180,E1 -31161.769,E2 -31161.769} C_VEL
LIN {X 0,Y 41.019,Z 366.561,A -85,B 0,C 180,E1 -31165.907,E2 -31165.907} C_VEL
LIN {X 0,Y 31.257,Z 373.719,A -85,B 0,C 180,E1 -31172.525,E2 -31172.525} C_VEL
LIN {X 0,Y 23.62,Z 378.557,A -85,B 0,C 180,E1 -31181.94,E2 -31181.94} C_VEL
LIN {X 0,Y 15.229,Z 383.711,A -85,B 0,C 180,E1 -31207.278,E2 -31207.278} C_VEL
LIN {X 0,Y 13.14,Z 387.853,A -85,B 0,C 180,E1 -31262.331,E2 -31262.331} C_VEL
LIN {X 0,Y 16.876,Z 389.49,A -85,B 0,C 180,E1 -31286.394,E2 -31286.394} C_VEL
LIN {X 0,Y 23.691,Z 390.875,A -85,B 0,C 180,E1 -31302.765,E2 -31302.765} C_VEL
LIN {X 0,Y 35.298,Z 391.798,A -85,B 0,C 180,E1 -31314.562,E2 -31314.562} C_VEL
LIN {X 0,Y 46.263,Z 391.5,A -85,B 0,C 180,E1 -31320.01,E2 -31320.01} C_VEL
LIN {X 0,Y 56.304,Z 390.328,A -85,B 0,C 180,E1 -31323.078,E2 -31323.078} C_VEL
LIN {X 0,Y 66.564,Z 388.266,A -85,B 0,C 180,E1 -31325.268,E2 -31325.268} C_VEL
LIN {X 0,Y 63.64,Z 389.004,A -85,B 0,C 180,E1 -31326.348,E2 -31326.348} C_VEL
LIN {X 0,Y 49.896,Z 391.363,A -85,B 0,C 180,E1 -31329.617,E2 -31329.617} C_VEL
LIN {X 0,Y 36.447,Z 392.197,A -85,B 0,C 180,E1 -31335.399,E2 -31335.399} C_VEL
LIN {X 0,Y 23.859,Z 391.452,A -85,B 0,C 180,E1 -31347.912,E2 -31347.912} C_VEL
LIN {X 0,Y 14.446,Z 389.194,A -85,B 0,C 180,E1 -31380.892,E2 -31380.892} C_VEL
LIN {X 0,Y 13.007,Z 387.427,A -85,B 0,C 180,E1 -31409.59,E2 -31409.59} C_VEL
LIN {X 0,Y 13.264,Z 386.352,A -85,B 0,C 180,E1 -31425.986,E2 -31425.986} C_VEL
LIN {X 0,Y 14.254,Z 384.439,A -85,B 0,C 180,E1 -31449.058,E2 -31449.058} C_VEL
LIN {X 0,Y 16.359,Z 382.263,A -85,B 0,C 180,E1 -31468.483,E2 -31468.483} C_VEL
LIN {X 0,Y 22.494,Z 378.028,A -85,B 0,C 180,E1 -31488.95,E2 -31488.95} C_VEL
LIN {X 0,Y 27.316,Z 375.117,A -85,B 0,C 180,E1 -31493.78,E2 -31493.78} C_VEL
LIN {X 0,Y 36.931,Z 368.739,A -85,B 0,C 180,E1 -31497.518,E2 -31497.518} C_VEL
LIN {X 0,Y 47.069,Z 360.525,A -85,B 0,C 180,E1 -31499.99,E2 -31499.99} C_VEL
LIN {X 0,Y 47.203,Z 359.967,A -85,B 0,C 180,E1 -31508.552,E2 -31508.552} C_VEL
LIN {X 0,Y 45.907,Z 361.321,A -85,B 0,C 180,E1 -31514.553,E2 -31514.553} C_VEL
LIN {X 0,Y 34.961,Z 369.892,A -85,B 0,C 180,E1 -31517.285,E2 -31517.285} C_VEL
LIN {X 0,Y 26.372,Z 375.41,A -85,B 0,C 180,E1 -31521.137,E2 -31521.137} C_VEL
LIN {X 0,Y 16.267,Z 380.82,A -85,B 0,C 180,E1 -31530.22,E2 -31530.22} C_VEL
LIN {X 0,Y 7.192,Z 385.075,A -85,B 0,C 180,E1 -31560.719,E2 -31560.719} C_VEL
LIN {X 0,Y 7.982,Z 388.276,A -85,B 0,C 180,E1 -31651.7,E2 -31651.7} C_VEL
LIN {X 0,Y 14.199,Z 389.868,A -85,B 0,C 180,E1 -31671.843,E2 -31671.843} C_VEL
LIN {X 0,Y 21.438,Z 391.035,A -85,B 0,C 180,E1 -31680.022,E2 -31680.022} C_VEL
LIN {X 0,Y 28.18,Z 391.709,A -85,B 0,C 180,E1 -31684.002,E2 -31684.002} C_VEL
LIN {X 0,Y 28.295,Z 391.754,A -85,B 0,C 180,E1 -31686.546,E2 -31686.546} C_VEL
LIN {X 0,Y 14.861,Z 390.192,A -85,B 0,C 180,E1 -31698.95,E2 -31698.95} C_VEL
LIN {X 0,Y 8.945,Z 388.805,A -85,B 0,C 180,E1 -31718.218,E2 -31718.218} C_VEL
LIN {X 0,Y 5.919,Z 386.965,A -85,B 0,C 180,E1 -31770.003,E2 -31770.003} C_VEL
LIN {X 0,Y 11.68,Z 383.293,A -85,B 0,C 180,E1 -31834.498,E2 -31834.498} C_VEL
LIN {X 0,Y 21.402,Z 378.46,A -85,B 0,C 180,E1 -31850.109,E2 -31850.109} C_VEL
LIN {X 0,Y 27.316,Z 375.117,A -85,B 0,C 180,E1 -31853.78,E2 -31853.78} C_VEL
LIN {X 0,Y 30.251,Z 376.852,A -85,B 0,C 180,E1 -31854.979,E2 -31854.979} C_VEL
LIN {X 0,Y 30.251,Z 600,A -85,B 0,C 180,E1 -31854.979,E2 -31854.979} C_VEL
LIN {X 0,Y 30.251,Z 600,A -85,B 0,C 180,E1 -31854.979,E2 -31854.979}

QRS_NEXT_CUT()

QRS_NEXT()
QRS_HOME()

END
